// Startable job contract processed by Worker.
INTERFACE I_Job EXTENDS I_Debug

// Called every worker cycle while Busy.
METHOD JobExecute
VAR_INPUT
END_VAR
END_METHOD

// Called once when the worker leaves Done.
METHOD JobExit
VAR_INPUT
END_VAR
END_METHOD

// Called once when the worker enters Init.
METHOD JobInit
VAR_INPUT
END_VAR
END_METHOD

END_INTERFACE

(* stored: Version 1.1.0.1
   Itf I_Job: Id {e5e86b3e-8f5d-4f0e-8f93-6a1bea47cd17}
   Method JobExecute: Id {9ac5d431-1fda-46e0-ab4e-6656d6c24d71}
   Method JobExit: Id {054d6bc8-13d0-47de-b56b-f58a14af1d76}
   Method JobInit: Id {f14910af-641c-4be5-ac57-b421cbbb9b13} *)
